// TIA Portal V19 export
DATA_BLOCK "ItemAlarmsOP"   // DB5
{ S7_Optimized_Access := 'TRUE' }
AUTHOR : FLA
FAMILY : UHT
VERSION : 1.0
// stored: AutoNumber false, MemoryReserve 0
   VAR
      Item : Array[1..32] of Bool;
   END_VAR
BEGIN
   // Item[1] : FB_FAULT_VALVE_01_01
   // Item[2] : FB_FAULT_VALVE_01_03
   // Item[3] : FB_FAULT_VALVE_01_04
   // Item[4] : FB_FAULT_VALVE_01_09
   // Item[5] : FB_FAULT_VALVE_01_11
   // Item[6] : FB_FAULT_VALVE_01_12
   // Item[7] : FB_FAULT_VALVE_01_13
   // Item[8] : FB_FAULT_VALVE_01_14
   // Item[9] : FB_FAULT_VALVE_01_15
   // Item[10] : FB_FAULT_MOTOR_01_39
   // Item[11] : FB_FAULT_MOTOR_01_30
   // Item[12] : FB_FAULT_VALVE_02_37
   // Item[13] : FB_FAULT_VALVE_02_38
   // Item[14] : FB_FAULT_VALVE_01_16
   // Item[15] : FB_FAULT_VALVE_01_17
   // Item[16] : FB_FAULT_VALVE_01_08
   // Item[17] : FB_FAULT_VALVE_01_19
   // Item[18] : FB_FAULT_VALVE_WATERPUMP
   // Item[19] : FB_FAULT_VALVE_09_04
   // Item[20] : FB_FAULT_VALVE_09_05
   // Item[21] : FB_FAULT_VALVE_09_06
   // Item[22] : FB_FAULT_VALVE_09_07
   // Item[23] : FB_FAULT_VALVE_09_08
   // Item[24] : FB_FAULT_VALVE_09_09
   // Item[25] : FB_FAULT_VALVE_09_10
   // Item[26] : FB_FAULT_VALVE_09_11
   // Item[27] : FB_FAULT_VALVE_09_12
   // Item[28] : FB_FAULT_VALVE_09_30
   // Item[29] : FB_FAULT_VALVE_09_31
   // Item[30] : DBX3_5
   // Item[31] : DBX3_6
   // Item[32] : DBX3_7
END_DATA_BLOCK
